// LS Electric XG5000 project: 16-46-3
// PLC NewPLC
// module base 0 slot 0: 입출력 모듈:XBC-DR14E (DC 24V 입력 8점, 릴레이 출력 6점)

PROGRAM NewProgram (task: 스캔 프로그램)

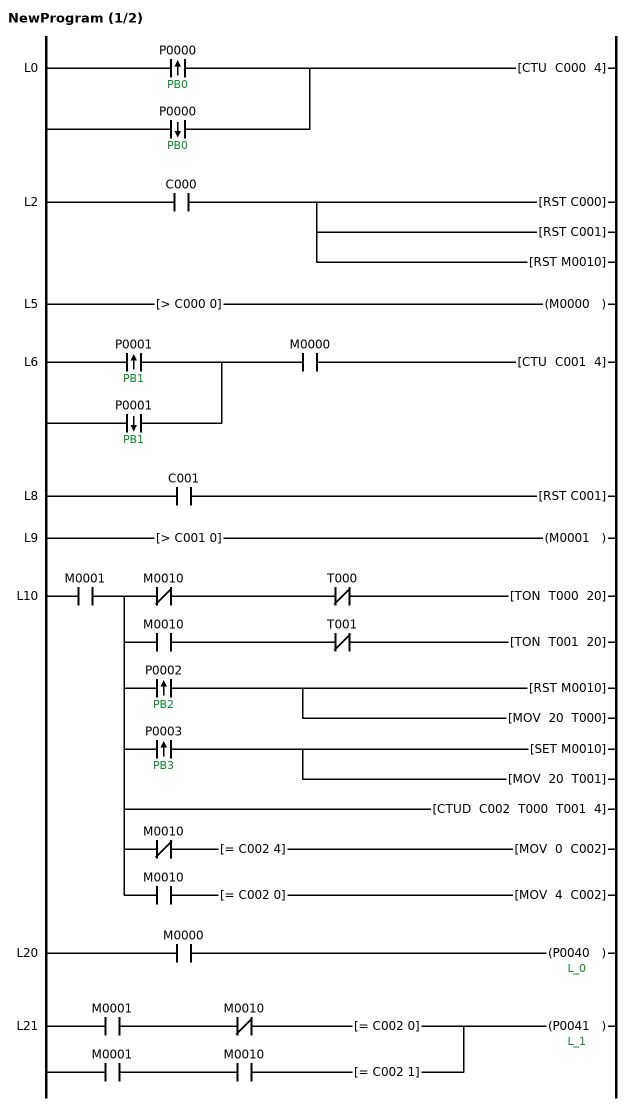
; L0
LOADP     P0000	// PB0
ORN       P0000	// PB0
CTU       C000 4
; L2
LOAD      C000
RST       C000
RST       C001
RST       M0010
; L5
LOAD>     C000 0
OUT       M0000
; L6
LOADP     P0001	// PB1
ORN       P0001	// PB1
AND       M0000
CTU       C001 4
; L8
LOAD      C001
RST       C001
; L9
LOAD>     C001 0
OUT       M0001
; L10
LOAD      M0001
MPUSH
AND NOT   M0010
AND NOT   T000
TON       T000 20
MLOAD
AND       M0010
AND NOT   T001
TON       T001 20
MLOAD
ANDP      P0002	// PB2
RST       M0010
MOV       20 T000
MLOAD
ANDP      P0003	// PB3
SET       M0010
MOV       20 T001
MLOAD
CTUD      C002 T000 T001 4
AND NOT   M0010
AND=      C002 4
MOV       0 C002
MPOP
AND       M0010
AND=      C002 0
MOV       4 C002
; L20
LOAD      M0000
OUT       P0040	// L_0
; L21
LOAD      M0001
AND NOT   M0010
AND=      C002 0
LOAD      M0001
AND       M0010
AND=      C002 1
OR LOAD
OUT       P0041	// L_1

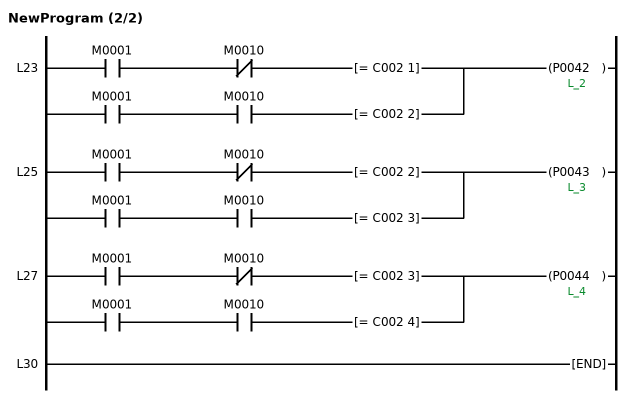
; L23
LOAD      M0001
AND NOT   M0010
AND=      C002 1
LOAD      M0001
AND       M0010
AND=      C002 2
OR LOAD
OUT       P0042	// L_2
; L25
LOAD      M0001
AND NOT   M0010
AND=      C002 2
LOAD      M0001
AND       M0010
AND=      C002 3
OR LOAD
OUT       P0043	// L_3
; L27
LOAD      M0001
AND NOT   M0010
AND=      C002 3
LOAD      M0001
AND       M0010
AND=      C002 4
OR LOAD
OUT       P0044	// L_4
; L30
END